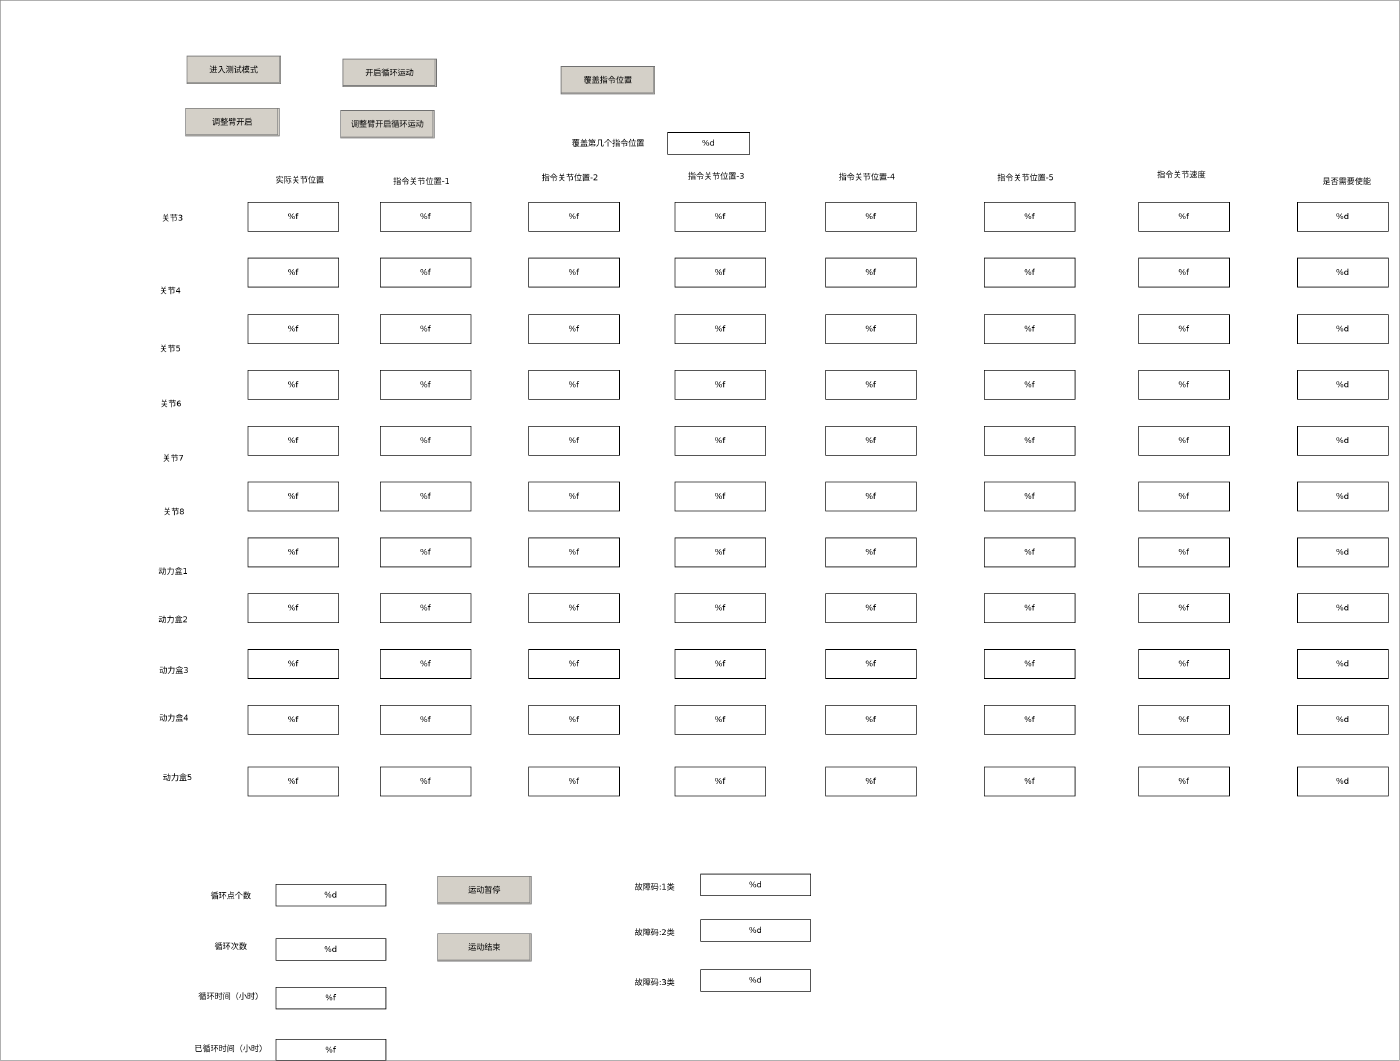
VISUALIZATION cycle_a3  // 1905x1445
    Button (254,76 128x38), "进入测试模式", colour toggle: g_cycleTest.m_enterCycleTestMode[3]
        toggle g_cycleTest.m_enterCycleTestMode[3]
    Button (466,80 128x38), "开启循环运动", colour toggle: g_cycleTest.m_startMotion[3]
        toggle g_cycleTest.m_startMotion[3]
    Label (501,233 145x28), "指令关节位置-1"
    Label (333,230 150x30), "实际关节位置"
    Rectangle (337,504 124x40), "%f", text variable: g_cycleTest.m_actJntPos[3][1]
    Label (162,283 145x28), "关节3"
    Label (159,382 145x28), "关节4"
    Label (159,461 145x28), "关节5"
    Label (160,536 145x28), "关节6"
    Label (163,610 145x28), "关节7"
    Label (164,683 145x28), "关节8"
    Label (163,764 145x28), "动力盒1"
    Label (163,830 145x28), "动力盒2"
    Label (169,1045 145x28), "动力盒5"
    Label (164,899 145x28), "动力盒3"
    Label (164,964 145x28), "动力盒4"
    Rectangle (337,580 124x40), "%f", text variable: g_cycleTest.m_actJntPos[3][2]
    Rectangle (337,656 124x40), "%f", text variable: g_cycleTest.m_actJntPos[3][3]
    Rectangle (337,732 124x40), "%f", text variable: g_cycleTest.m_actJntPos[3][4]
    Rectangle (337,808 124x40), "%f", text variable: g_cycleTest.m_actJntPos[3][5]
    Rectangle (337,884 124x40), "%f", text variable: g_cycleTest.m_actJntPos[3][6]
    Rectangle (337,960 124x40), "%f", text variable: g_cycleTest.m_actJntPos[3][7]
    Rectangle (337,1044 124x40), "%f", text variable: g_cycleTest.m_actJntPos[3][8]
    Rectangle (337,275 124x40), "%f", text variable: g_cycleTest.m_actJntPosSetup[3][3]
    Rectangle (337,351 124x40), "%f", text variable: g_cycleTest.m_actJntPosSetup[3][4]
    Rectangle (337,428 124x40), "%f", text variable: g_cycleTest.m_actJntPosSetup[3][5]
    Rectangle (517,275 124x40), "%f", text variable: g_cycleTest.m_targetJntPosSetup[3,1][3]
        OnMouseClick: write the text variable via Default
    Rectangle (517,351 124x40), "%f", text variable: g_cycleTest.m_targetJntPosSetup[3,1][4]
        OnMouseClick: write the text variable via Default
    Rectangle (517,428 124x40), "%f", text variable: g_cycleTest.m_targetJntPosSetup[3,1][5]
        OnMouseClick: write the text variable via Default
    Rectangle (517,504 124x40), "%f", text variable: g_cycleTest.m_targetJntPos[3,1][1]
        OnMouseClick: write the text variable via Default
    Rectangle (517,580 124x40), "%f", text variable: g_cycleTest.m_targetJntPos[3,1][2]
        OnMouseClick: write the text variable via Default
    Rectangle (517,656 124x40), "%f", text variable: g_cycleTest.m_targetJntPos[3,1][3]
        OnMouseClick: write the text variable via Default
    Rectangle (517,732 124x40), "%f", text variable: g_cycleTest.m_targetJntPos[3,1][4]
        OnMouseClick: write the text variable via Default
    Rectangle (517,808 124x40), "%f", text variable: g_cycleTest.m_targetJntPos[3,1][5]
        OnMouseClick: write the text variable via Default
    Rectangle (517,884 124x40), "%f", text variable: g_cycleTest.m_targetJntPos[3,1][6]
        OnMouseClick: write the text variable via Default
    Rectangle (517,960 124x40), "%f", text variable: g_cycleTest.m_targetJntPos[3,1][7]
        OnMouseClick: write the text variable via Default
    Rectangle (517,1044 124x40), "%f", text variable: g_cycleTest.m_targetJntPos[3,1][8]
        OnMouseClick: write the text variable via Default
    Label (703,228 145x28), "指令关节位置-2"
    Rectangle (719,275 124x40), "%f", text variable: g_cycleTest.m_targetJntPosSetup[3,2][3]
        OnMouseClick: write the text variable via Default
    Rectangle (719,351 124x40), "%f", text variable: g_cycleTest.m_targetJntPosSetup[3,2][4]
        OnMouseClick: write the text variable via Default
    Rectangle (719,428 124x40), "%f", text variable: g_cycleTest.m_targetJntPosSetup[3,2][5]
        OnMouseClick: write the text variable via Default
    Rectangle (719,504 124x40), "%f", text variable: g_cycleTest.m_targetJntPos[3,2][1]
        OnMouseClick: write the text variable via Default
    Rectangle (719,580 124x40), "%f", text variable: g_cycleTest.m_targetJntPos[3,2][2]
        OnMouseClick: write the text variable via Default
    Rectangle (719,656 124x40), "%f", text variable: g_cycleTest.m_targetJntPos[3,2][3]
        OnMouseClick: write the text variable via Default
    Rectangle (719,732 124x40), "%f", text variable: g_cycleTest.m_targetJntPos[3,2][4]
        OnMouseClick: write the text variable via Default
    Rectangle (719,808 124x40), "%f", text variable: g_cycleTest.m_targetJntPos[3,2][5]
        OnMouseClick: write the text variable via Default
    Rectangle (719,884 124x40), "%f", text variable: g_cycleTest.m_targetJntPos[3,2][6]
        OnMouseClick: write the text variable via Default
    Rectangle (719,960 124x40), "%f", text variable: g_cycleTest.m_targetJntPos[3,2][7]
        OnMouseClick: write the text variable via Default
    Rectangle (719,1044 124x40), "%f", text variable: g_cycleTest.m_targetJntPos[3,2][8]
        OnMouseClick: write the text variable via Default
    Label (902,226 145x28), "指令关节位置-3"
    Rectangle (918,275 124x40), "%f", text variable: g_cycleTest.m_targetJntPosSetup[3,3][3]
        OnMouseClick: write the text variable via Default
    Rectangle (918,351 124x40), "%f", text variable: g_cycleTest.m_targetJntPosSetup[3,3][4]
        OnMouseClick: write the text variable via Default
    Rectangle (918,428 124x40), "%f", text variable: g_cycleTest.m_targetJntPosSetup[3,3][5]
        OnMouseClick: write the text variable via Default
    Rectangle (918,504 124x40), "%f", text variable: g_cycleTest.m_targetJntPos[3,3][1]
        OnMouseClick: write the text variable via Default
    Rectangle (918,580 124x40), "%f", text variable: g_cycleTest.m_targetJntPos[3,3][2]
        OnMouseClick: write the text variable via Default
    Rectangle (918,656 124x40), "%f", text variable: g_cycleTest.m_targetJntPos[3,3][3]
        OnMouseClick: write the text variable via Default
    Rectangle (918,732 124x40), "%f", text variable: g_cycleTest.m_targetJntPos[3,3][4]
        OnMouseClick: write the text variable via Default
    Rectangle (918,808 124x40), "%f", text variable: g_cycleTest.m_targetJntPos[3,3][5]
        OnMouseClick: write the text variable via Default
    Rectangle (918,884 124x40), "%f", text variable: g_cycleTest.m_targetJntPos[3,3][6]
        OnMouseClick: write the text variable via Default
    Rectangle (918,960 124x40), "%f", text variable: g_cycleTest.m_targetJntPos[3,3][7]
        OnMouseClick: write the text variable via Default
    Rectangle (918,1044 124x40), "%f", text variable: g_cycleTest.m_targetJntPos[3,3][8]
        OnMouseClick: write the text variable via Default
    Label (1107,227 145x28), "指令关节位置-4"
    Rectangle (1123,275 124x40), "%f", text variable: g_cycleTest.m_targetJntPosSetup[3,4][3]
        OnMouseClick: write the text variable via Default
    Rectangle (1123,351 124x40), "%f", text variable: g_cycleTest.m_targetJntPosSetup[3,4][4]
        OnMouseClick: write the text variable via Default
    Rectangle (1123,428 124x40), "%f", text variable: g_cycleTest.m_targetJntPosSetup[3,4][5]
        OnMouseClick: write the text variable via Default
    Rectangle (1123,504 124x40), "%f", text variable: g_cycleTest.m_targetJntPos[3,4][1]
        OnMouseClick: write the text variable via Default
    Rectangle (1123,580 124x40), "%f", text variable: g_cycleTest.m_targetJntPos[3,4][2]
        OnMouseClick: write the text variable via Default
    Rectangle (1123,656 124x40), "%f", text variable: g_cycleTest.m_targetJntPos[3,4][3]
        OnMouseClick: write the text variable via Default
    Rectangle (1123,732 124x40), "%f", text variable: g_cycleTest.m_targetJntPos[3,4][4]
        OnMouseClick: write the text variable via Default
    Rectangle (1123,808 124x40), "%f", text variable: g_cycleTest.m_targetJntPos[3,4][5]
        OnMouseClick: write the text variable via Default
    Rectangle (1123,884 124x40), "%f", text variable: g_cycleTest.m_targetJntPos[3,4][6]
        OnMouseClick: write the text variable via Default
    Rectangle (1123,960 124x40), "%f", text variable: g_cycleTest.m_targetJntPos[3,4][7]
        OnMouseClick: write the text variable via Default
    Rectangle (1123,1044 124x40), "%f", text variable: g_cycleTest.m_targetJntPos[3,4][8]
        OnMouseClick: write the text variable via Default
    Label (1323,228 145x28), "指令关节位置-5"
    Rectangle (1339,275 124x40), "%f", text variable: g_cycleTest.m_targetJntPosSetup[3,5][3]
        OnMouseClick: write the text variable via Default
    Rectangle (1339,351 124x40), "%f", text variable: g_cycleTest.m_targetJntPosSetup[3,5][4]
        OnMouseClick: write the text variable via Default
    Rectangle (1339,428 124x40), "%f", text variable: g_cycleTest.m_targetJntPosSetup[3,5][5]
        OnMouseClick: write the text variable via Default
    Rectangle (1339,504 124x40), "%f", text variable: g_cycleTest.m_targetJntPos[3,5][1]
        OnMouseClick: write the text variable via Default
    Rectangle (1339,580 124x40), "%f", text variable: g_cycleTest.m_targetJntPos[3,5][2]
        OnMouseClick: write the text variable via Default
    Rectangle (1339,656 124x40), "%f", text variable: g_cycleTest.m_targetJntPos[3,5][3]
        OnMouseClick: write the text variable via Default
    Rectangle (1339,732 124x40), "%f", text variable: g_cycleTest.m_targetJntPos[3,5][4]
        OnMouseClick: write the text variable via Default
    Rectangle (1339,808 124x40), "%f", text variable: g_cycleTest.m_targetJntPos[3,5][5]
        OnMouseClick: write the text variable via Default
    Rectangle (1339,884 124x40), "%f", text variable: g_cycleTest.m_targetJntPos[3,5][6]
        OnMouseClick: write the text variable via Default
    Rectangle (1339,960 124x40), "%f", text variable: g_cycleTest.m_targetJntPos[3,5][7]
        OnMouseClick: write the text variable via Default
    Rectangle (1339,1044 124x40), "%f", text variable: g_cycleTest.m_targetJntPos[3,5][8]
        OnMouseClick: write the text variable via Default
    Button (252,147 128x38), "调整臂开启", colour toggle: g_cycleTest.m_enterCycleTestModeSetup[3]
        toggle g_cycleTest.m_enterCycleTestModeSetup[3]
    Button (463,150 128x38), "调整臂开启循环运动", colour toggle: g_cycleTest.m_startMotionSetup[3]
        toggle g_cycleTest.m_startMotionSetup[3]
    Label (1535,224 145x28), "指令关节速度"
    Rectangle (1549,275 124x40), "%f", text variable: g_cycleTest.m_targetJntVelSetup[3][3]
        OnMouseClick: write the text variable via Default
    Rectangle (1549,351 124x40), "%f", text variable: g_cycleTest.m_targetJntVelSetup[3][4]
        OnMouseClick: write the text variable via Default
    Rectangle (1549,428 124x40), "%f", text variable: g_cycleTest.m_targetJntVelSetup[3][5]
        OnMouseClick: write the text variable via Default
    Rectangle (1549,504 124x40), "%f", text variable: g_cycleTest.m_targetJntVelN8[3][1]
        OnMouseClick: write the text variable via Default
    Rectangle (1549,580 124x40), "%f", text variable: g_cycleTest.m_targetJntVelN8[3][2]
        OnMouseClick: write the text variable via Default
    Rectangle (1549,656 124x40), "%f", text variable: g_cycleTest.m_targetJntVelN8[3][3]
        OnMouseClick: write the text variable via Default
    Rectangle (1549,732 124x40), "%f", text variable: g_cycleTest.m_targetJntVelN8[3][4]
        OnMouseClick: write the text variable via Default
    Rectangle (1549,808 124x40), "%f", text variable: g_cycleTest.m_targetJntVelN8[3][5]
        OnMouseClick: write the text variable via Default
    Rectangle (1549,884 124x40), "%f", text variable: g_cycleTest.m_targetJntVelN8[3][6]
        OnMouseClick: write the text variable via Default
    Rectangle (1549,960 124x40), "%f", text variable: g_cycleTest.m_targetJntVelN8[3][7]
        OnMouseClick: write the text variable via Default
    Rectangle (1549,1044 124x40), "%f", text variable: g_cycleTest.m_targetJntVelN8[3][8]
        OnMouseClick: write the text variable via Default
    Button (763,90 128x38), "覆盖指令位置", colour toggle: g_cycleTest.m_coverCmdPos[3]
        tap g_cycleTest.m_coverCmdPos[3]
    Rectangle (908,180 112x30), "%d", text variable: g_cycleTest.m_pntIdForCoverCmd[3]
        OnMouseClick: write the text variable via Default
    Label (755,181 145x28), "覆盖第几个指令位置"
    Label (239,1205 150x30), "循环点个数"
    Rectangle (375,1204 150x30), "%d", text variable: g_cycleTest.m_pointSum[3]
        OnMouseClick: write the text variable via Default
    Rectangle (375,1278 150x30), "%d", text variable: g_cycleTest.m_curCycleNum[3]
        OnMouseClick: write the text variable via Default
    Label (239,1274 150x30), "循环次数"
    Button (595,1193 128x38), "运动暂停", colour toggle: g_cycleTest.m_pause[3]
        toggle g_cycleTest.m_pause[3]
    Button (595,1271 128x38), "运动结束", colour toggle: g_cycleTest.m_finish[3]
        tap g_cycleTest.m_finish[3]
    Rectangle (375,1344 150x30), "%f", text variable: g_cycleTest.m_tgtCycleTime[3]
        OnMouseClick: write the text variable via Default
    Label (239,1342 150x30), "循环时间（小时）"
    Rectangle (375,1415 150x30), "%f", text variable: g_cycleTest.m_curCycleTime[3]
        OnMouseClick: write the text variable via Default
    Label (239,1413 150x30), "已循环时间（小时）"
    Label (1760,232 145x30), "是否需要使能"
    Rectangle (1765,275 124x40), "%d", text variable: g_cycleTest.m_jntEnableSetup[3][3]
        OnMouseClick: write the text variable via Default
    Rectangle (1765,351 124x40), "%d", text variable: g_cycleTest.m_jntEnableSetup[3][4]
        OnMouseClick: write the text variable via Default
    Rectangle (1765,428 124x40), "%d", text variable: g_cycleTest.m_jntEnableSetup[3][5]
        OnMouseClick: write the text variable via Default
    Rectangle (1765,504 124x40), "%d", text variable: g_cycleTest.m_jntEnable[3][1]
        OnMouseClick: write the text variable via Default
    Rectangle (1765,580 124x40), "%d", text variable: g_cycleTest.m_jntEnable[3][2]
        OnMouseClick: write the text variable via Default
    Rectangle (1765,656 124x40), "%d", text variable: g_cycleTest.m_jntEnable[3][3]
        OnMouseClick: write the text variable via Default
    Rectangle (1765,732 124x40), "%d", text variable: g_cycleTest.m_jntEnable[3][4]
        OnMouseClick: write the text variable via Default
    Rectangle (1765,808 124x40), "%d", text variable: g_cycleTest.m_jntEnable[3][5]
        OnMouseClick: write the text variable via Default
    Rectangle (1765,884 124x40), "%d", text variable: g_cycleTest.m_jntEnable[3][6]
        OnMouseClick: write the text variable via Default
    Rectangle (1765,960 124x40), "%d", text variable: g_cycleTest.m_jntEnable[3][7]
        OnMouseClick: write the text variable via Default
    Rectangle (1765,1044 124x40), "%d", text variable: g_cycleTest.m_jntEnable[3][8]
        OnMouseClick: write the text variable via Default
    Rectangle (953,1190 150x30), "%d", text variable: GVL_interactUI.g_errIdType1
        OnMouseClick: write the text variable via Default
    Label (816,1193 150x30), "故障码:1类"
    Rectangle (953,1252 150x30), "%d", text variable: GVL_interactUI.g_errIdType2
        OnMouseClick: write the text variable via Default
    Label (816,1255 150x30), "故障码:2类"
    Rectangle (953,1320 150x30), "%d", text variable: GVL_interactUI.g_errIdType3
        OnMouseClick: write the text variable via Default
    Label (816,1323 150x30), "故障码:3类"
END_VISUALIZATION

(* stored: Version 1.1.0.1, ProductVersion 3.1.4024.11
   Visu cycle_a3: Id {55d79b45-4f42-4fc5-b554-fed32a543f42} *)
